# EPICS substitutions: EPICS7/IOCs/loopback/loopbackApp/Db/user.substitutions
# SPDX-FileCopyrightText: 2006 Argonne National Laboratory
#
# SPDX-License-Identifier: EPICS

# Example substitutions file

file "db/circle.db" {
    { user = "ys" }
}

file "db/dbExample1.db" {
    { user = "ys" }
}

file db/dbExample2.db {
    pattern { user, no, scan }
        { "ys", 1, "1 second" }
        { "ys", 2, "2 second" }
        { "ys", 3, "5 second" }
}
